PROGRAM MAIN
VAR
	bEnable : BOOL;
	bStart : BOOL;
	nINT : INT := -32768;
	nUINT : UINT := 65535;
	fREAL : REAL := 255.255;
	nFloatConversion : INT;
	fFloatConversion : LREAL;
	nIntConversion : INT;
	fIntConversion : LREAL;
	

	
END_VAR

bEnable := bStart;
fFloatConversion := INT_TO_LREAL(nFloatConversion);
nIntConversion := LREAL_TO_INT(fIntConversion);

END_PROGRAM

(* stored: Version 1.1.0.1, ProductVersion 3.1.4024.12
   POU MAIN: Id {0fe40e25-b51c-485e-ad15-ae3716e33560}, SpecialFunc None *)
